// TIA Portal V17 export
// export: Created 2022-07-20T06:59:36.3661916Z, ExportSetting WithDefaults, DisplayName Totally Integrated Automation Portal, DisplayVersion V17, DisplayName TIA Portal Openness, DisplayVersion V17, DisplayName TIA Portal Version Control Interface, DisplayVersion V17, DisplayName SINAMICS Startdrive Advanced, DisplayVersion V17, DisplayName SINAMICS Startdrive G130, G150, S120, S150, SINAMICS MV, S210, DisplayVersion V17, DisplayName SINAMICS Startdrive G110M, G120, G120C, G120D, G120P, G115D, DisplayVersion V17, DisplayName STEP 7 Professional, DisplayVersion V17, DisplayName STEP 7 Safety, DisplayVersion V17, DisplayName WinCC Advanced, DisplayVersion V17
FUNCTION_BLOCK "FB10001_PulseControl"   // FB10001, LAD
TITLE = FB10001_PulseControl
{ S7_Optimized_Access := 'TRUE' }
AUTHOR : Jonathan
FAMILY : 1000x_SYSTEM
VERSION : 1.0
// Release note : 
// 1.0 - Feature developped
// stored: AutoNumber false, IsIECCheckEnabled false, IsRetainMemResEnabled false, MemoryReserve 100, SetENOAutomatically false, UDAEnableTagReadback false
   VAR_INPUT
      Time_On : Time;
      Time_Off : Time;
      Signal : Bool;
   END_VAR
   VAR_OUTPUT
      SignalPulsed : Bool;
   END_VAR
   VAR
      TON_On { S7_SetPoint := 'True'} : TON_TIME;
      TON_Off { S7_SetPoint := 'True'} : TON_TIME;
   END_VAR
BEGIN

REGION Network 1 (SCL): Pulse Control Management
   #TON_On(IN := #TON_Off.Q,
            PT := #Time_On);

   #TON_Off(IN := #Signal AND NOT #TON_On.Q,
            PT := #Time_Off);

   #SignalPulsed := #TON_Off.Q;
END_REGION
END_FUNCTION_BLOCK
